// TIA Portal project "Endüstriyel Kapı" (V17)

(* hardware
DEVICE "S71500/ET200MP-Station_1"  S7-1500 station
   slot 0: "Profilschiene_0"  6ES7 590-1***0-0AA0
   slot 1: "PLC_1"  CPU 1511-1 PN  6ES7 511-1AK00-0AB0  V1.8
   slot 2: "AI 8xU/I/RTD/TC ST_1"  AI 8xU/I/RTD/TC ST  6ES7 531-7KF00-0AB0  V2.0
   slot 3: "AI 8xU/I/RTD/TC ST_2"  AI 8xU/I/RTD/TC ST  6ES7 531-7KF00-0AB0  V2.0
   slot 4: "AI 8xU/I/RTD/TC ST_3"  AI 8xU/I/RTD/TC ST  6ES7 531-7KF00-0AB0  V2.0
   slot 5: "AI 8xU/I/RTD/TC ST_4"  AI 8xU/I/RTD/TC ST  6ES7 531-7KF00-0AB0  V2.0
   slot 6: "DI 16x24VDC BA_1"  DI 16x24VDC BA  6ES7 521-1BH10-0AA0  V1.0
*)

// ===== PLC "PLC_1"  CPU 1511-1 PN =====

VAR_GLOBAL   // PLC tag table "Standard-Variablentabelle"
   "AÇMA (MÜHÜRLÜ)" AT %E0.0 : Bool;
   "KAPAMA (MÜHÜRLÜ)(1)" AT %E0.1 : Bool;
   "AÇMA (KESİK)" AT %I0.2 : Bool;
   "KAPAMA (KESİK)" AT %I0.3 : Bool;
   "KAPI KAPALI SENSÖRÜ" AT %I0.4 : Bool;
   "KAPI AÇIK SENSÖR" AT %I0.5 : Bool;
   "YAKINLIK SENSÖRÜ" AT %I0.6 : Bool;
   "ACİL STOP" AT %I0.7 : Bool;
   "KAPI AÇMA" AT %Q0.0 : Bool;
   "KAPI KAPAMA" AT %Q0.1 : Bool;
   "UYARI IŞIK" AT %Q0.2 : Bool;
   "KAPI AÇMA Y.K" AT %M0.0 : Bool;
   "KAPI KAPAMA Y.K" AT %M0.1 : Bool;
   "Tag_1" AT %M50.0 : Bool;
   "Tag_2" AT %M50.1 : Bool;
   "Tag_3" AT %M50.2 : Bool;
   "Tag_4" AT %M50.3 : Bool;
   "Tag_5" AT %M50.4 : Bool;
   "Tag_6" AT %M50.5 : Bool;
   "5sn BEKLEME" AT %T37 : Timer;
   "Clock_Byte" AT %MB40 : Byte;
   "Clock_10Hz" AT %M40.0 : Bool;
   "Clock_5Hz" AT %M40.1 : Bool;
   "Clock_2.5Hz" AT %M40.2 : Bool;
   "Clock_2Hz" AT %M40.3 : Bool;
   "Clock_1.25Hz" AT %M40.4 : Bool;
   "Clock_1Hz" AT %M40.5 : Bool;
   "Clock_0.625Hz" AT %M40.6 : Bool;
   "Clock_0.5Hz" AT %M40.7 : Bool;
   "Tag_8" AT %M50.6 : Bool;
END_VAR

// folder: System blocks/Program resources

DATA_BLOCK "T37"   // DB2
{ S7_Optimized_Access := 'TRUE' }
AUTHOR : Simatic
FAMILY : IEC
NAME : IEC_TMR
VERSION : 1.0
// stored: InstanceOfName IEC_TIMER
"IEC_TIMER"
BEGIN
END_DATA_BLOCK

// folder: (top level)

FUNCTION "MHJ-PLC-Lab-Function-S71500" : Void   // FC9000, SCL
{ S7_Optimized_Access := 'TRUE' }
VERSION : 0.1
   VAR_TEMP
      Value : Byte;
      ForCounter : Int;
   END_VAR
   VAR CONSTANT
      Value_01_DW : DWord := 16#1223_5486;
      Value_02_DW : DWord := 16#A6C9_D1F5;
   END_VAR
BEGIN

   #Value:=PEEK(area := 16#82,
        dbNumber := 0,
        byteOffset := 511);
   #Value := #Value + 1;

   POKE(area := 16#82,
        dbNumber := 0,
        byteOffset := 511,
        value := #Value);

   POKE(area := 16#82,
        dbNumber := 0,
        byteOffset := 1016,
        value := #Value_01_DW);
   POKE(area := 16#82,
        dbNumber := 0,
        byteOffset := 1020,
        value := #Value_02_DW);

   FOR #ForCounter := 0 TO 63 DO
       #Value:=PEEK(area := 16#1,
            dbNumber := 0,
            byteOffset := #ForCounter);
       POKE(area := 16#81,
            dbNumber := 0,
            byteOffset := #ForCounter,
            value := #Value);
   END_FOR;
   #Value := PEEK(area := 16#1,
                  dbNumber := 0,
                  byteOffset := 512);
   POKE(area := 16#82,
        dbNumber := 0,
        byteOffset := 512,
        value := #Value);
END_FUNCTION

ORGANIZATION_BLOCK "Main"   // OB1, LAD, ProgramCycle
TITLE = "Main Program Sweep (Cycle)"
{ S7_Optimized_Access := 'TRUE' }
VERSION : 0.1
   VAR_INPUT
      Initial_Call : Bool;   // Initial call of this OB
      Remanence : Bool;   // =True, if remanent data are available
   END_VAR
   VAR_TEMP   // added for the SCL form of the ladder/FBD networks
      _w1 : Bool;
   END_VAR
BEGIN

REGION Network 1
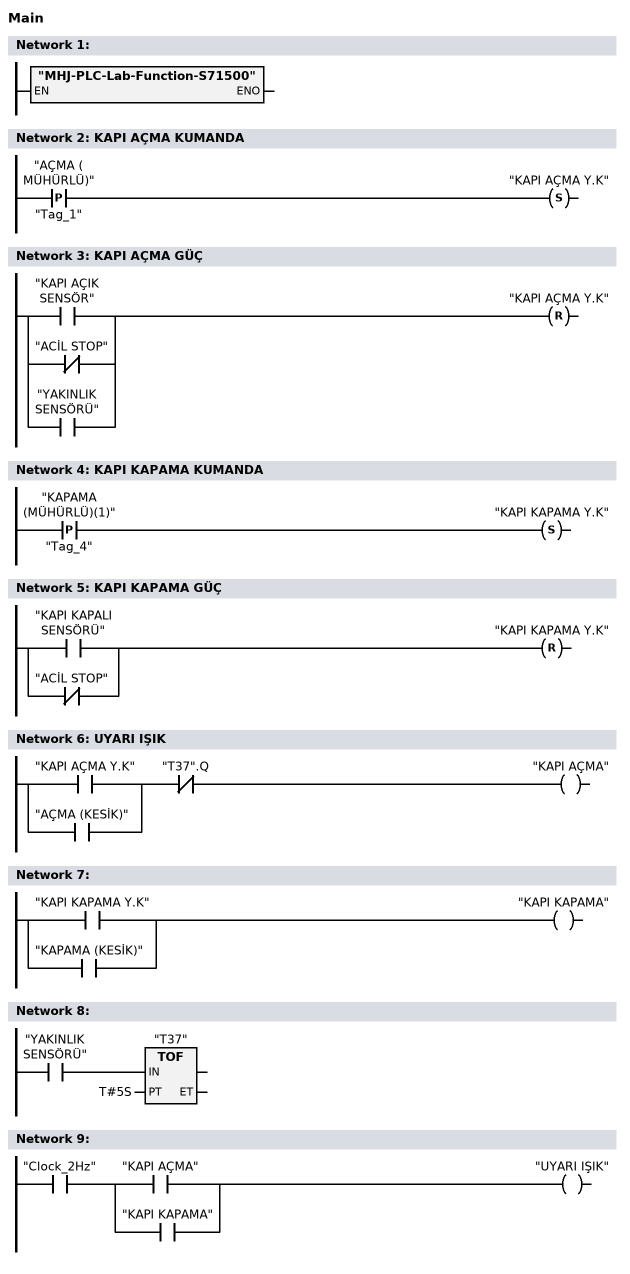
   RUNG wire#powerrail
      "MHJ-PLC-Lab-Function-S71500"()
   END_RUNG
   // the same network as SCL:
   "MHJ-PLC-Lab-Function-S71500"();
END_REGION

REGION Network 2: KAPI AÇMA KUMANDA
   RUNG wire#powerrail
      P_Contact(operand := "AÇMA (MÜHÜRLÜ)", bit := "Tag_1")
      S_Coil( "KAPI AÇMA Y.K" )
   END_RUNG
   // the same network as SCL:
   #_w1 := "AÇMA (MÜHÜRLÜ)" AND NOT "Tag_1";   // rising edge of "AÇMA (MÜHÜRLÜ)"
   "Tag_1" := "AÇMA (MÜHÜRLÜ)";
   IF #_w1 THEN "KAPI AÇMA Y.K" := TRUE; END_IF;
END_REGION

REGION Network 3: KAPI AÇMA GÜÇ
   RUNG wire#powerrail
      Contact( "KAPI AÇIK SENSÖR" )
      wire#w1
      R_Coil( "KAPI AÇMA Y.K" )
   END_RUNG
   RUNG wire#powerrail
      I_Contact( "ACİL STOP" )
   END_RUNG wire#w1
   RUNG wire#powerrail
      Contact( "YAKINLIK SENSÖRÜ" )
   END_RUNG wire#w1
   // the same network as SCL:
   IF "KAPI AÇIK SENSÖR" OR NOT "ACİL STOP" OR "YAKINLIK SENSÖRÜ" THEN "KAPI AÇMA Y.K" := FALSE; END_IF;
END_REGION

REGION Network 4: KAPI KAPAMA KUMANDA
   RUNG wire#powerrail
      P_Contact(operand := "KAPAMA (MÜHÜRLÜ)(1)", bit := "Tag_4")
      S_Coil( "KAPI KAPAMA Y.K" )
   END_RUNG
   // the same network as SCL:
   #_w1 := "KAPAMA (MÜHÜRLÜ)(1)" AND NOT "Tag_4";   // rising edge of "KAPAMA (MÜHÜRLÜ)(1)"
   "Tag_4" := "KAPAMA (MÜHÜRLÜ)(1)";
   IF #_w1 THEN "KAPI KAPAMA Y.K" := TRUE; END_IF;
END_REGION

REGION Network 5: KAPI KAPAMA GÜÇ
   RUNG wire#powerrail
      Contact( "KAPI KAPALI SENSÖRÜ" )
      wire#w1
      R_Coil( "KAPI KAPAMA Y.K" )
   END_RUNG
   RUNG wire#powerrail
      I_Contact( "ACİL STOP" )
   END_RUNG wire#w1
   // the same network as SCL:
   IF "KAPI KAPALI SENSÖRÜ" OR NOT "ACİL STOP" THEN "KAPI KAPAMA Y.K" := FALSE; END_IF;
END_REGION

REGION Network 6: UYARI IŞIK
   RUNG wire#powerrail
      Contact( "KAPI AÇMA Y.K" )
      wire#w1
      I_Contact( "T37".Q )
      Coil( "KAPI AÇMA" )
   END_RUNG
   RUNG wire#powerrail
      Contact( "AÇMA (KESİK)" )
   END_RUNG wire#w1
   // the same network as SCL:
   "KAPI AÇMA" := ("KAPI AÇMA Y.K" OR "AÇMA (KESİK)") AND NOT "T37".Q;
END_REGION

REGION Network 7
   RUNG wire#powerrail
      Contact( "KAPI KAPAMA Y.K" )
      wire#w1
      Coil( "KAPI KAPAMA" )
   END_RUNG
   RUNG wire#powerrail
      Contact( "KAPAMA (KESİK)" )
   END_RUNG wire#w1
   // the same network as SCL:
   "KAPI KAPAMA" := "KAPI KAPAMA Y.K" OR "KAPAMA (KESİK)";
END_REGION

REGION Network 8
   "T37".TOF(IN := "YAKINLIK SENSÖRÜ", PT := T#5S);
END_REGION

REGION Network 9
   RUNG wire#powerrail
      Contact( "Clock_2Hz" )
      wire#w1
      Contact( "KAPI AÇMA" )
      wire#w2
      Coil( "UYARI IŞIK" )
   END_RUNG
   RUNG wire#w1
      Contact( "KAPI KAPAMA" )
   END_RUNG wire#w2
   // the same network as SCL:
   "UYARI IŞIK" := "Clock_2Hz" AND ("KAPI AÇMA" OR "KAPI KAPAMA");
END_REGION
END_ORGANIZATION_BLOCK